// Mitsubishi GX Works2 project: MODBUS_RTU_SLAVE   PLC: FX3U/FX3UC

PROGRAM MAIN
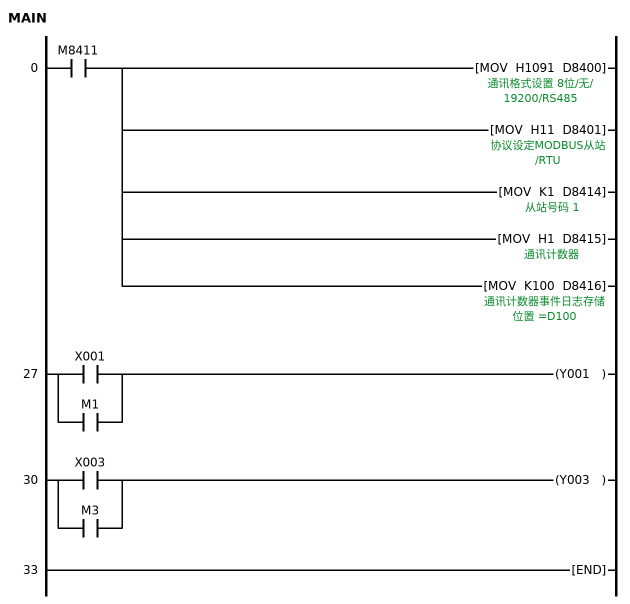
0     LD      M8411
      MOV     H1091 D8400  ; 通讯格式设置 8位/无/19200/RS485
      MOV     H11 D8401  ; 协议设定MODBUS从站/RTU
      MOV     K1 D8414  ; 从站号码 1
      MOV     H1 D8415  ; 通讯计数器
      MOV     K100 D8416  ; 通讯计数器事件日志存储位置 =D100
27    LD      X001
      OR      M1
      OUT     Y001
30    LD      X003
      OR      M3
      OUT     Y003
33    END
END_PROGRAM
